(* CoDeSys 2.3 library: TcIoFunctions.lb6 *)
(* Libraries: STANDARD.LB6 5.6.98 12:03:02 *)

(* Data type *)
TYPE ST_KL1501InData :
STRUCT
	iState		: USINT;
	iDummy		: USINT;
	arrDataIn	: ARRAY[0..1] OF UINT;
END_STRUCT
END_TYPE

(* Data type *)
TYPE ST_KL1501OutData :
STRUCT
	iCtrl		: USINT;
	iDummy		: USINT;
	arrDataOut	: ARRAY[0..1] OF UINT;
END_STRUCT
END_TYPE

(* Data type *)
TYPE ST_KL27x1InData :
STRUCT
	iState		: USINT;
	iDummy		: USINT;
	iDataIn		: INT;
END_STRUCT
END_TYPE

(* Data type *)
TYPE ST_KL27x1OutData :
STRUCT
	iCtrl		: USINT;
	iDummy		: USINT;
	iDataOut	: INT;
END_STRUCT
END_TYPE

(* Data type *)
TYPE ST_KL3208InData :
STRUCT
	iState		: USINT;
	iDummy		: USINT;
	iDataIn		: INT;
END_STRUCT
END_TYPE

(* Data type *)
TYPE ST_KL3208OutData :
STRUCT
	iCtrl		: USINT;
	iDummy		: USINT;
	iDataOut	: INT;
END_STRUCT
END_TYPE

(* Data type *)
TYPE ST_KL320xInData :
STRUCT
	iState		: USINT;
	iDummy		: USINT;
	iDataIn		: INT;
END_STRUCT
END_TYPE

(* Data type *)
TYPE ST_KL320xOutData :
STRUCT
	iCtrl		: USINT;
	iDummy		: USINT;
	iDataOut	: INT;
END_STRUCT
END_TYPE

(* Data type *)
TYPE ST_KL3228InData :
STRUCT
	iState		: USINT;
	iDummy		: USINT;
	iDataIn		: INT;
END_STRUCT
END_TYPE

(* Data type *)
TYPE ST_KL3228OutData :
STRUCT
	iCtrl		: USINT;
	iDummy		: USINT;
	iDataOut	: INT;
END_STRUCT
END_TYPE

(* POU F_GetVersionTcIoFunctions, ST *)
FUNCTION F_GetVersionTcIoFunctions : UINT	(*Gets the library version info *)
VAR_INPUT
	nVersionElement		:	INT;
END_VAR
(*
	Possible nVersionElement parameter:
	1	:	major number
	2	:	minor number
	3	:	revision number
*)
VAR
END_VAR
(* Version history:
Date		|	Version	|	created with	|	Author		|	Remark
dd.mm.yyyy
-----------------------------------------------------------------------------------------------------------------------------------------------------------------------------------------------------------------
26.01.2016	|	1.0.0	|	TC 2.11 B2252	|	Peter S.  	|	first TC 2.11 release Folder K-Bus Terminals FB_KL1501Config, FB_KL27x1Config, FB_KL3208Config, FB_KL320xConfig, FB_KL3228Config;
*)	
CASE nVersionElement OF
1:	(* major number *)
	F_GetVersionTcIoFunctions := 1;
2:	(* minor number *)
	F_GetVersionTcIoFunctions := 0;
3:	(* revision number *)
	F_GetVersionTcIoFunctions := 0;
ELSE
	F_GetVersionTcIoFunctions := 16#FFFF;
END_CASE
END_FUNCTION

(* POU FB_KL1501Config, ST *)
FUNCTION_BLOCK FB_KL1501Config
VAR_INPUT
	bConfigurate			: BOOL; 		(*Rising edge starts configuration including read-configuration afterwards*)
	bReadConfig				: BOOL;			(*Rising edge reads the actual configuration*)
	iSetCounterType			: INT;			(*Counter-type to be set, see table*)
	bSetBackwardCounting	: BOOL;			(*Select backward-counting*)
	tTimeout				: TIME :=t#5s;	(*Time-out-time for Reading/Configuration - initially set to 5s*)
END_VAR
VAR_OUTPUT
	bBusy					: BOOL;			(*Reading or configuration is in progress*)
	bError					: BOOL;			(*Error while reading/configuration*)
	iErrorId				: UDINT;		(*Id of the last upcoming error*)
	iState					: USINT;		(*As long as the funcion-block is not busy, this variable shows the state of the terminal, otherwise it is 0*)
	iDataIn0				: UINT;			(*As long as the funcion-block is not busy, this variable shows the dataIn0 of the terminal, otherwise it keeps the value previous to reding/configuration*)
	iDataIn1				: UINT;			(*As long as the funcion-block is not busy, this variable shows the dataIn1 of the terminal, otherwise it keeps the value previous to reding/configuration*)
	iDataIn					: UDINT;		(*iDataIn1 and IDataIn0 put together as an UDINT, with iDataIn1 as High-Integer*)
	iTerminalType			: WORD;			(*Terminal-type-number, in this case 3228*)
	iSpecialType			: WORD;			(*Sub-type-number*)
	iFirmwareVersion		: WORD;			(*Firmware in ASCII-code*)
	sDescription			: STRING;		(*Terminal-type, special-type and firmware-version as readable text*)
	sCounterType			: STRING;		(*Text-description of entered counter-type*)
	bBackwardCounting		: BOOL;			(*TRUE: Backward-counting was selected*)
END_VAR
VAR
	rtRead					: R_TRIG;
	rtSet					: R_TRIG;
	bSetReq					: BOOL;
	tonTimeout				: TON;
	iStep					: INT;
	bSetConfigError			: BOOL;
	wReg32					: WORD;
	wSetReg32				: WORD;
	wFirmware				: WORD;
	pFirmware				: POINTER TO WORD;
	sFirmware				: STRING(2);
	iDataIn0Saved			: UINT;
	iDataIn1Saved			: UINT;
END_VAR
VAR_IN_OUT
	stInData   				: ST_KL1501InData;	(* Process image of the inputs. *)
	stOutData 				: ST_KL1501OutData;	(* Process image of the outputs. *)
END_VAR
tonTimeout	(PT:=tTimeout);
IF	tonTimeout.Q	THEN
	bError			:= TRUE;
	iErrorId		:= 16#8001;
	iStep			:= 0;
END_IF

rtSet	(CLK:=bConfigurate);
rtRead	(CLK:=bReadConfig);

IF	(rtSet.Q OR rtRead.Q)	AND NOT bBusy THEN
	bBusy			:= TRUE;
	bError			:= FALSE;
	iErrorId		:= 0;
	iDataIn0Saved	:= stInData.arrDataIn[0];
	iDataIn1Saved	:= stInData.arrDataIn[1];
	tonTimeout.IN	:= TRUE;
	iStep			:= 10;
	IF	rtSet.Q	THEN
		bSetReq	:= TRUE;
	END_IF
END_IF

IF bBusy THEN
	iDataIn0	:= iDataIn0Saved;
	iDataIn1	:= iDataIn1Saved;
	iState		:= 0;
ELSE
	iDataIn0	:= stInData.arrDataIn[0];
	iDataIn1	:= stInData.arrDataIn[1];
	iState		:= stInData.iState;
END_IF

iDataIn	:= UINT_TO_UDINT(iDataIn0)+(UINT_TO_UDINT(iDataIn1)*65536);

CASE iStep OF

0:	(*idle*)
	bBusy				:= FALSE;
	bSetReq				:= FALSE;
	tonTimeout.IN		:= FALSE;

10:	(*Klemmentyp (Kl32xx) auslesen: Register 8*)
	stOutData.iCtrl	:= 16#88;	(*Register 8 Lesen*)

	IF stInData.iState = 16#88 THEN
		iTerminalType	:= UINT_TO_WORD(stInData.arrDataIn[0]);
		iStep:=20;
	END_IF

20:	(*Spezialtyp (Kl1501-yyy) auslesen: Register 29*)
	stOutData.iCtrl	:= 16#9D;	(*Register 29 Lesen*)

	IF stInData.iState = 16#9D THEN
		iSpecialType	:= UINT_TO_WORD(stInData.arrDataIn[0]);
		iStep:=30;
	END_IF

30:	(*Firmware auslesen: Register 9*)
	stOutData.iCtrl	:= 16#89;	(*Register 9 Lesen*)

	IF stInData.iState = 16#89 THEN
		iFirmwareVersion:= UINT_TO_WORD(stInData.arrDataIn[0]);
		(*Umwandlung in STRING*)
		wFirmware		:= iFirmwareVersion;
		wFirmware		:= ROR(wFirmware,8);(*Reihenfolge der beiden Zeichen der Firmware tauschen*)
		pFirmware		:= ADR(sFirmware);	(*Einen Pointer auf den Info-String (Ausgang) legen*)
		pFirmware^		:= wFirmware;		(*Diesen Adressbereich mit dem richtig getauschen Wert beschreiben - damit ist auch der String beschrieben*)

		sDescription	:= CONCAT('Terminal ',WORD_TO_STRING(iTerminalType));

		CASE LEN(WORD_TO_STRING(iSpecialType)) OF
			1: sDescription	:= CONCAT(sDescription,'-000');
			2: sDescription	:= CONCAT(sDescription,'-00');
			3: sDescription	:= CONCAT(sDescription,'-0');
		ELSE
			sDescription	:= CONCAT(sDescription,'-');
		END_CASE

		sDescription	:= CONCAT(sDescription,WORD_TO_STRING(iSpecialType));
		sDescription	:= CONCAT(sDescription,' / Firmware ');
		sDescription	:= CONCAT(sDescription,sFirmware);

		IF bSetReq	THEN
			iStep:=100;
		ELSE
			iStep:=150;
		END_IF
	END_IF

	(*Falscher Klemmentyp angeschlossen, Konfiguration vorzeitig abbrechen*)
	IF (iTerminalType <> 1501)	THEN
		bError		:= TRUE;
		iErrorId	:= 16#8002;
		iStep		:= 160;
	END_IF
(*-----------------------------------------------------------------*)

100:(*jetzige Sensoreinstellung lesen: Register 32*)
	stOutData.iCtrl	:= 16#A0;	(*Register 32 Lesen*)

	IF stInData.iState = 16#A0 THEN
		wReg32			:= UINT_TO_WORD(stInData.arrDataIn[0]);
		A_SetConfigTable;			(*entsprechende Einstellungen vornehmen*)
		iStep:=110;
		IF	bSetConfigError	THEN
			iStep:=150;
		END_IF
	END_IF

110:(*Codewort Register 31 setzen: 16#1235 -> Schreibschutz aufheben*)
	stOutData.iCtrl	:= 16#DF;	(*Register 31 beschreiben*)
	stOutData.arrDataOut[0]	:= 16#1235;	(*Nutzdaten: Codewort*)

	IF stInData.iState = 16#9F THEN
		stOutData.iCtrl	:= 16#9F;	(*Register 31 Auslesen*)
		iStep:=120;
	END_IF

120:(*Bestätigung Codewort gesetzt erfragen*)
	IF	stInData.arrDataIn[0]	= 16#1235	THEN
		iStep:=130;
	END_IF

130:(*Nun Register 32 mit dem neuen Wert beschreiben*)
	stOutData.iCtrl	:= 16#E0;	(*Register 32 beschreiben*)
	stOutData.arrDataOut[0]	:= WORD_TO_UINT(wSetReg32);

	IF stInData.iState = 16#A0 THEN
		iStep:=140;
	END_IF

140:(*Codewort Register 31 löschen: 16#0000 -> Schreibschutz setzen*)
	stOutData.iCtrl	:= 16#DF;	(*Register 31 beschreiben*)
	stOutData.arrDataOut[0]	:= 16#0000;

	IF stInData.iState = 16#9F THEN
		iStep:=150;
	END_IF

150:(*nach erfolgter Parametrierung Sensoreinstellung lesen: Register 32*)
	stOutData.iCtrl	:= 16#A0;	(*Register 32 Lesen*)

	IF stInData.iState = 16#A0 THEN
		wReg32			:= UINT_TO_WORD(stInData.arrDataIn[0]);
		A_ReadConfigTable;
		iStep:=160;
	END_IF

160:(*Registerkommunikation beenden*)
	stOutData.iCtrl	:= 0; (*auch alle anderen Steuerbits mit ablöschen*)
	(*Rückmeldeabfrage Prozessdatenaustausch (Bit7) noch aktiv? *)
	(*alle anderen Bits könnten durch einen bestimmten Signalpegel gesetzt sein *)
	IF stInData.iState.7 = FALSE THEN
		iStep:=0;
	END_IF

END_CASE
END_FUNCTION_BLOCK
ACTION A_ReadConfigTable:
CASE (wReg32 AND 2#11100000000) OF	(*Check sensor-type via bits 8-10*)
	2#00100000000: sCounterType:='32-bit forward-backward-counter';
	2#01000000000: sCounterType:='Two 16-bit-forward-counter';
	2#10000000000: sCounterType:='32-bit gated forward-counter - Gate low inhibits';
	2#10100000000: sCounterType:='32-bit gated forward-counter - Gate high inhibits';
ELSE
	sCounterType:='Unknown';
	bError		:= TRUE;
	iErrorId	:= 16#8011;
END_CASE

bBackwardCounting:=wReg32.11;
END_ACTION
ACTION A_SetConfigTable:
bSetConfigError	:= FALSE;

wSetReg32:=wReg32 AND 2#1111000011111111;(*First clear the characteristical bits (8-11)*)

CASE iSetCounterType OF	(*Then set the counter-type via the bits 8-11*)

	0:	wSetReg32:=wSetReg32 OR 2#00100000000;(*32-bit forward-backward-counter*)
		wSetReg32.11:=bSetBackwardCounting;

	1:	wSetReg32:=wSetReg32 OR 2#01000000000;(*Two 16-bit-forward-counter*)
		wSetReg32.11:=bSetBackwardCounting;

	2:	wSetReg32:=wSetReg32 OR 2#10000000000;(*32-bit gated forward-counter - Gate low inhibits*)
		wSetReg32.11:=bSetBackwardCounting;

	3:	wSetReg32:=wSetReg32 OR 2#10100000000;(*32-bit gated forward-counter - Gate high inhibits*)
		wSetReg32.11:=bSetBackwardCounting;
ELSE
	bSetConfigError	:= TRUE;
	bError			:= TRUE;
	iErrorId		:= 16#8010;
END_CASE
END_ACTION

(* POU FB_KL27x1Config, ST *)
FUNCTION_BLOCK FB_KL27x1Config
VAR_INPUT
	bConfigurate			: BOOL; 		(*Rising edge starts configuration including read-configuration afterwards*)
	bReadConfig				: BOOL;			(*Rising edge reads the actual configuration*)
	bSetDimRampAbsolute		: BOOL;			(*FALSE: ramp-time refers to a step from 0..100%, TRUE: ramp-time refers to a step to the next value*)
	iSetRampTime			: INT;			(*Ramp-time to be set, see table*)
	bSetWatchdogDisable		: BOOL;			(*TRUE disables the watchdog for fieldbus-communication*)
	iSetWatchdogTimeout		: UINT;			(*Watchdog-time in 10ms-units*)
	iSetTimeoutOnValue		: UINT;			(*Value to be set, if timeout occurs and lamp was previously turned on*)
	iSetTimeoutOffValue		: UINT;			(*Value to be set, if timeout occurs and lamp was previously turned off*)
	iSetDimmerMode			: INT;			(*Dimmer-mode to be set, see table*)
	bSetOnAfterShortCircuit	: BOOL;			(*Selects, if the lamp has to be turned on after short-circuit*)
	bSetLineFrequency60Hz	: BOOL;			(*FALSE sets the line-frequency to 50Hz, TRUE to 60Hz*)
	tTimeout				: TIME :=t#5s;	(*Time-out-time for Reading/Configuration - initially set to 5s*)
END_VAR
VAR_OUTPUT
	bBusy					: BOOL;			(*Reading or configuration is in progress*)
	bError					: BOOL;			(*Error while reading/configuration*)
	iErrorId				: UDINT;		(*Id of the last upcoming error*)
	iState					: USINT;		(*As long as the funcion-block is not busy, this variable shows the state of the terminal, otherwise it is 0*)
	iTerminalType			: WORD;			(*Terminal-type-number, e.g. 2751*)
	iSpecialType			: WORD;			(*Sub-type-number*)
	iFirmwareVersion		: WORD;			(*Firmware in ASCII-code*)
	sDescription			: STRING;		(*Terminal-type, special-type and firmware-version as readable text*)

	bDimRampAbsolute		: BOOL;			(*TRUE: Dimramp was set to absolute - FALSE Dimramp was set to relative*)
	sRampTime				: STRING;		(*Ramp-time, which was set, according to the table*)
	bWatchdogDisable		: BOOL;			(*TRUE: Watchdog was disabled*)
	tWatchdogTimeout		: TIME;			(*Entered Watchdog-time*)
	iTimeoutOnValue			: UINT;			(*Timeout on-value, which was set*)
	iTimeoutOffValue		: UINT;			(*Timeout off-value, which was set*)
	sDimmerMode				: STRING;		(*Dimmer-mode, which was selected*)
	sAfterShortCircuit		: STRING;		(*Selected behaviour after short-circuit - on or off*)
	sLineFrequency			: STRING;		(*Selected line-frequency - 50 or 60 Hz*)
END_VAR
VAR
	rtRead					: R_TRIG;
	rtSet					: R_TRIG;
	bSetReq					: BOOL;
	tonTimeout				: TON;
	iStep					: INT;
	bSetConfigError			: BOOL;
	wReg32					: WORD;
	wSetReg32				: WORD;
	wReg35					: WORD;
	wSetReg35				: WORD;
	wReg36					: WORD;
	wSetReg36				: WORD;
	wReg37					: WORD;
	wSetReg37				: WORD;
	wReg38					: WORD;
	wSetReg38				: WORD;
	wReg39					: WORD;
	wSetReg39				: WORD;
	wReg40					: WORD;
	wSetReg40				: WORD;
	wReg41					: WORD;
	wSetReg41				: WORD;
	wFirmware				: WORD;
	pFirmware				: POINTER TO WORD;
	sFirmware				: STRING(2);
END_VAR
VAR_IN_OUT
	stInData   				: ST_KL27x1InData;	(* Process image of the inputs. *)
	stOutData 				: ST_KL27x1OutData;	(* Process image of the outputs. *)
END_VAR
tonTimeout	(PT:=tTimeout);
IF	tonTimeout.Q	THEN
	bError			:= TRUE;
	iErrorId		:= 16#8001;
	iStep			:= 0;
END_IF

rtSet	(CLK:=bConfigurate);
rtRead	(CLK:=bReadConfig);

IF	(rtSet.Q OR rtRead.Q)	AND NOT bBusy THEN
	bBusy			:= TRUE;
	bError			:= FALSE;
	iErrorId		:= 0;
	tonTimeout.IN	:= TRUE;
	iStep			:= 10;
	IF	rtSet.Q	THEN
		bSetReq	:= TRUE;
	END_IF
END_IF

IF bBusy THEN
	iState		:= 0;
ELSE
	iState		:= stInData.iState;
END_IF


CASE iStep OF

0:	(*idlde*)
	bBusy				:= FALSE;
	bSetReq				:= FALSE;
	tonTimeout.IN		:= FALSE;

10:	(*Klemmentyp (Kl27xx) auslesen: Register 8*)
	stOutData.iCtrl	:= 16#88;	(*Register 8 Lesen*)

	IF stInData.iState = 16#88 THEN
		iTerminalType	:= INT_TO_WORD(stInData.iDataIn);
		iStep:=20;
	END_IF

20:	(*Spezialtyp (Kl27xx-yyy) auslesen: Register 29*)
	stOutData.iCtrl	:= 16#9D;	(*Register 29 Lesen*)

	IF stInData.iState = 16#9D THEN
		iSpecialType	:= INT_TO_WORD(stInData.iDataIn);
		iStep:=30;
	END_IF

30:	(*Firmware auslesen: Register 9*)
	stOutData.iCtrl	:= 16#89;	(*Register 9 Lesen*)

	IF stInData.iState = 16#89 THEN
		iFirmwareVersion:= INT_TO_WORD(stInData.iDataIn);
		(*Umwandlung in STRING*)
		wFirmware		:= iFirmwareVersion;
		wFirmware		:= ROR(wFirmware,8);(*Reihenfolge der beiden Zeichen der Firmware tauschen*)
		pFirmware		:= ADR(sFirmware);	(*Einen Pointer auf den Info-String (Ausgang) legen*)
		pFirmware^		:= wFirmware;		(*Diesen Adressbereich mit dem richtig getauschen Wert beschreiben - damit ist auch der String beschrieben*)

		sDescription	:= CONCAT('Terminal ',WORD_TO_STRING(iTerminalType));

		CASE LEN(WORD_TO_STRING(iSpecialType)) OF
			1: sDescription	:= CONCAT(sDescription,'-000');
			2: sDescription	:= CONCAT(sDescription,'-00');
			3: sDescription	:= CONCAT(sDescription,'-0');
		ELSE
			sDescription	:= CONCAT(sDescription,'-');
		END_CASE

		sDescription	:= CONCAT(sDescription,WORD_TO_STRING(iSpecialType));
		sDescription	:= CONCAT(sDescription,' / Firmware ');
		sDescription	:= CONCAT(sDescription,sFirmware);

		IF bSetReq	THEN
			iStep:=100;
		ELSE
			iStep:=150;
		END_IF
	END_IF

	(*Falscher Klemmentyp angeschlossen, Konfiguration vorzeitig abbrechen*)
	IF ((iTerminalType <> 2751)	AND (iTerminalType <> 2761))	THEN
		bError		:= TRUE;
		iErrorId	:= 16#8002;
		iStep		:= 160;
	END_IF

(*-----------------------------------------------------------------*)

100:(*jetzige Sensoreinstellung lesen: Register 32*)
	stOutData.iCtrl	:= 16#A0;	(*Register 32 Lesen*)

	IF stInData.iState = 16#A0 THEN
		wReg32			:= INT_TO_WORD(stInData.iDataIn);
		A_SetConfigTable;			(*entsprechende Einstellungen vornehmen*)
		iStep:=110;
		IF	bSetConfigError	THEN
			iStep:=150;
		END_IF
	END_IF

110:(*Codewort Register 31 setzen: 16#1235 -> Schreibschutz aufheben*)
	stOutData.iCtrl	:= 16#DF;	(*Register 31 beschreiben*)
	stOutData.iDataOut	:= 16#1235;	(*Nutzdaten: Codewort*)

	IF stInData.iState = 16#9F THEN
		stOutData.iCtrl	:= 16#9F;	(*Register 31 Auslesen*)
		iStep:=120;
	END_IF

120:(*Bestätigung Codewort gesetzt erfragen*)
	IF	stInData.iDataIn	= 16#1235	THEN
		iStep:=130;
	END_IF

130:(*Register 32 mit dem neuen Wert beschreiben*)
	stOutData.iCtrl	:= 16#E0;	(*Register 32 beschreiben*)
	stOutData.iDataOut	:= WORD_TO_INT(wSetReg32);

	IF stInData.iState = 16#A0 THEN
		iStep:=131;
	END_IF

131:(*Register 35 mit dem neuen Wert beschreiben*)
	stOutData.iCtrl	:= 16#E3;	(*Register 35 beschreiben*)
	stOutData.iDataOut	:= WORD_TO_INT(wSetReg35);

	IF stInData.iState = 16#A3 THEN
		iStep:=132;
	END_IF

132:(*Register 36 mit dem neuen Wert beschreiben*)
	stOutData.iCtrl	:= 16#E4;	(*Register 36 beschreiben*)
	stOutData.iDataOut	:= WORD_TO_INT(wSetReg36);

	IF stInData.iState = 16#A4 THEN
		iStep:=133;
	END_IF

133:(*Register 37 mit dem neuen Wert beschreiben*)
	stOutData.iCtrl	:= 16#E5;	(*Register 37 beschreiben*)
	stOutData.iDataOut	:= WORD_TO_INT(wSetReg37);

	IF stInData.iState = 16#A5 THEN
		iStep:=134;
	END_IF

134:(*Register 38 mit dem neuen Wert beschreiben*)
	stOutData.iCtrl	:= 16#E6;	(*Register 38 beschreiben*)
	stOutData.iDataOut	:= WORD_TO_INT(wSetReg38);

	IF stInData.iState = 16#A6 THEN
		iStep:=135;
	END_IF

135:(*Register 39 mit dem neuen Wert beschreiben*)
	stOutData.iCtrl	:= 16#E7;	(*Register 39 beschreiben*)
	stOutData.iDataOut	:= WORD_TO_INT(wSetReg39);

	IF stInData.iState = 16#A7 THEN
		iStep:=136;
	END_IF

136:(*Register 40 mit dem neuen Wert beschreiben*)
	stOutData.iCtrl	:= 16#E8;	(*Register 40 beschreiben*)
	stOutData.iDataOut	:= WORD_TO_INT(wSetReg40);

	IF stInData.iState = 16#A8 THEN
		iStep:=137;
	END_IF

137:(*Register 41 mit dem neuen Wert beschreiben*)
	stOutData.iCtrl	:= 16#E9;	(*Register 41 beschreiben*)
	stOutData.iDataOut	:= WORD_TO_INT(wSetReg41);

	IF stInData.iState = 16#A9 THEN
		iStep:=140;
	END_IF

140:(*Codewort Register 31 löschen: 16#0000 -> Schreibschutz setzen*)
	stOutData.iCtrl	:= 16#DF;	(*Register 31 beschreiben*)
	stOutData.iDataOut	:= 16#0000;

	IF stInData.iState = 16#9F THEN
		iStep:=150;
	END_IF

150:(*nach erfolgter Parametrierung Konfiguration lesen: Register 32*)
	stOutData.iCtrl	:= 16#A0;	(*Register 32 Lesen*)

	IF stInData.iState = 16#A0 THEN
		wReg32			:= INT_TO_WORD(stInData.iDataIn);
		iStep:=151;
	END_IF

151:(*nach erfolgter Parametrierung Konfiguration lesen: Register 35*)
	stOutData.iCtrl	:= 16#A3;	(*Register 35 Lesen*)

	IF stInData.iState = 16#A3 THEN
		wReg35			:= INT_TO_WORD(stInData.iDataIn);
		iStep:=152;
	END_IF

152:(*nach erfolgter Parametrierung Konfiguration lesen: Register 36*)
	stOutData.iCtrl	:= 16#A4;	(*Register 36 Lesen*)

	IF stInData.iState = 16#A4 THEN
		wReg36			:= INT_TO_WORD(stInData.iDataIn);
		iStep:=153;
	END_IF

153:(*nach erfolgter Parametrierung Konfiguration lesen: Register 37*)
	stOutData.iCtrl	:= 16#A5;	(*Register 37 Lesen*)

	IF stInData.iState = 16#A5 THEN
		wReg37			:= INT_TO_WORD(stInData.iDataIn);
		iStep:=154;
	END_IF

154:(*nach erfolgter Parametrierung Konfiguration lesen: Register 38*)
	stOutData.iCtrl	:= 16#A6;	(*Register 38 Lesen*)

	IF stInData.iState = 16#A6 THEN
		wReg38			:= INT_TO_WORD(stInData.iDataIn);
		iStep:=155;
	END_IF

155:(*nach erfolgter Parametrierung Konfiguration lesen: Register 39*)
	stOutData.iCtrl	:= 16#A7;	(*Register 39 Lesen*)

	IF stInData.iState = 16#A7 THEN
		wReg39			:= INT_TO_WORD(stInData.iDataIn);
		iStep:=156;
	END_IF

156:(*nach erfolgter Parametrierung Konfiguration lesen: Register 40*)
	stOutData.iCtrl	:= 16#A8;	(*Register 40 Lesen*)

	IF stInData.iState = 16#A8 THEN
		wReg40			:= INT_TO_WORD(stInData.iDataIn);
		iStep:=157;
	END_IF


157:(*nach erfolgter Parametrierung Konfiguration lesen: Register 41*)
	stOutData.iCtrl	:= 16#A9;	(*Register 41 Lesen*)

	IF stInData.iState = 16#A9 THEN
		wReg41			:= INT_TO_WORD(stInData.iDataIn);
		A_ReadConfigTable;
		iStep:=160;
	END_IF


160:(*Registerkommunikation beenden*)
	stOutData.iCtrl	:= 0; (*auch alle anderen Steuerbits mit ablöschen*)
	(*Rückmeldeabfrage Prozessdatenaustausch (Bit7) noch aktiv? *)
	(*alle anderen Bits könnten durch einen bestimmten Signalpegel gesetzt sein *)
	IF stInData.iState.7 = FALSE THEN
		iStep:=0;
	END_IF

END_CASE
END_FUNCTION_BLOCK
ACTION A_ReadConfigTable:
bWatchdogDisable	:= wReg32.2;
bDimRampAbsolute	:= wReg32.3;


CASE wReg35 OF
	0:	sRampTime	:= '50 ms';
	1:	sRampTime	:= '100 ms';
	2:	sRampTime	:= '200 ms';
	3:	sRampTime	:= '500 ms';
	4:	sRampTime	:= '1 s';
	5:	sRampTime	:= '2 s';
	6:	sRampTime	:= '5 s';
	7:	sRampTime	:= '10 s';
ELSE
	sRampTime	:= 'unknown register-entry';
	bError		:= TRUE;
	iErrorId	:= 16#801A;
END_CASE


tWatchdogTimeout	:= WORD_TO_TIME(wReg36)*10;
iTimeoutOnValue		:= wReg37;
iTimeoutOffValue	:= wReg38;


CASE wReg39 OF
	0:	sDimmerMode	:= '0 - Automatic recognition';
	1:	sDimmerMode	:= '1 - Trailing phase angle';
	2:	sDimmerMode	:= '2 - Leading phase angle';
	3:	sDimmerMode	:= '3 - Rectifier mode, positive';
	4:	sDimmerMode	:= '4 - Rectifier mode, negative';
ELSE
	sDimmerMode	:= 'unknown register-entry';
	bError		:= TRUE;
	iErrorId	:= 16#801B;
END_CASE


CASE wReg40 OF
	0:	sAfterShortCircuit := 'Off';
	1:	sAfterShortCircuit := 'On';
ELSE
	sAfterShortCircuit	:= 'unknown register-entry';
	bError				:= TRUE;
	iErrorId			:= 16#801C;
END_CASE


CASE wReg41 OF
	0:	sLineFrequency := '50 Hz';
	1:	sLineFrequency := '60 Hz';
ELSE
	sLineFrequency	:= 'unknown register-entry';
	bError			:= TRUE;
	iErrorId		:= 16#801D;
END_CASE
END_ACTION
ACTION A_SetConfigTable:
bSetConfigError	:= FALSE;

wSetReg32	:= wReg32	AND 2#1111111111110011;(*Clear bits 2 and 3 of Reg32*)
wSetReg32.2	:= bSetWatchdogDisable;
wSetReg32.3	:= bSetDimRampAbsolute;

CASE iSetRampTime OF
	0:	wSetReg35	:= 0;		(*50 ms*)
	1:	wSetReg35	:= 1;		(*100 ms*)
	2:	wSetReg35	:= 2;		(*200 ms*)
	3:	wSetReg35	:= 3;		(*500 ms*)
	4:	wSetReg35	:= 4;		(*1 s*)
	5:	wSetReg35	:= 5;		(*2 s*)
	6:	wSetReg35	:= 6;		(*5 s*)
	7:	wSetReg35	:= 7;		(*10 s*)
ELSE
	bSetConfigError	:= TRUE;
	bError			:= TRUE;
	iErrorId		:= 16#8018;
END_CASE


wSetReg36	:=	UINT_TO_WORD(iSetWatchdogTimeout);
wSetReg37	:=	UINT_TO_WORD(iSetTimeoutOnValue);
wSetReg38	:=	UINT_TO_WORD(iSetTimeoutOffValue);


CASE iSetDimmerMode OF
	0:	wSetReg39	:= 0;		(*automatic recognition*)
	1:	wSetReg39	:= 1;		(*trailing phase angle*)
	2:	wSetReg39	:= 2;		(*leading phase angle*)
	3:	wSetReg39	:= 3;		(*Rectifier mode, positive*)
	4:	wSetReg39	:= 4;		(*Rectifier mode, negative*)
ELSE
	bSetConfigError	:= TRUE;
	bError			:= TRUE;
	iErrorId		:= 16#8019;
END_CASE

IF	bSetOnAfterShortCircuit	THEN
		wSetReg40	:= 1;
ELSE	wSetReg40	:= 0;
END_IF

IF	bSetLineFrequency60Hz	THEN
		wSetReg41	:= 1;
ELSE	wSetReg41	:= 0;
END_IF
END_ACTION

(* POU FB_KL3208Config, ST *)
FUNCTION_BLOCK FB_KL3208Config
VAR_INPUT
	bConfigurate		: BOOL; 		(*Rising edge starts configuration including read-configuration afterwards*)
	bReadConfig			: BOOL;			(*Rising edge reads the actual configuration*)
	iSetSensorType		: INT;			(*Sensor-type to be set, see table*)
	tTimeout			: TIME :=t#5s;	(*Time-out-time for Reading/Configuration - initially set to 5s*)
END_VAR
VAR_OUTPUT
	bBusy				: BOOL;			(*Reading or configuration is in progress*)
	bError				: BOOL;			(*Error while reading/configuration*)
	iErrorId			: UDINT;		(*Id of the last upcoming error*)
	iState				: USINT;		(*As long as the funcion-block is not busy, this variable shows the state of the terminal, otherwise it is 0*)
	iDataIn				: INT;			(*As long as the funcion-block is not busy, this variable shows the dataIn of the terminal, otherwise it keeps the value previous to reding/configuration*)
	iTerminalType		: WORD;			(*Terminal-type-number, in this case 3208*)
	iSpecialType		: WORD;			(*Sub-type-number*)
	iFirmwareVersion	: WORD;			(*Firmware in ASCII-code*)
	sDescription		: STRING;		(*Terminal-type, special-type and firmware-version as readable text*)
	sSensorType			: STRING;		(*Text-description of entered sensor-type*)
END_VAR
VAR
	rtRead				: R_TRIG;
	rtSet				: R_TRIG;
	bSetReq				: BOOL;
	tonTimeout			: TON;
	iStep				: INT;
	bSetConfigError		: BOOL;
	wReg32				: WORD;
	wSetReg32			: WORD;
	wReg39				: WORD;
	wSetReg39			: WORD;
	wFirmware			: WORD;
	pFirmware			: POINTER TO WORD;
	sFirmware			: STRING(2);
	iDataInSaved		: INT;
END_VAR
VAR_IN_OUT
	stInData   			: ST_KL3208InData;	(* Process image of the inputs. *)
	stOutData 			: ST_KL3208OutData;	(* Process image of the outputs. *)
END_VAR
tonTimeout	(PT:=tTimeout);
IF	tonTimeout.Q	THEN
	bError			:= TRUE;
	iErrorId		:= 16#8001;
	iStep			:= 0;
END_IF

rtSet	(CLK:=bConfigurate);
rtRead	(CLK:=bReadConfig);

IF	(rtSet.Q OR rtRead.Q)	AND NOT bBusy THEN
	bBusy			:= TRUE;
	bError			:= FALSE;
	iErrorId		:= 0;
	iDataInSaved	:= stInData.iDataIn;
	tonTimeout.IN	:= TRUE;
	iStep			:= 10;
	IF	rtSet.Q	THEN
		bSetReq	:= TRUE;
	END_IF
END_IF

IF bBusy THEN
	iDataIn		:= iDataInSaved;
	iState		:= 0;
ELSE
	iDataIn		:= stInData.iDataIn;
	iState		:= stInData.iState;
END_IF


CASE iStep OF

0:	(*idle*)
	bBusy				:= FALSE;
	bSetReq				:= FALSE;
	tonTimeout.IN		:= FALSE;

10:	(*Klemmentyp (Kl32xx) auslesen: Register 8*)
	stOutData.iCtrl	:= 16#88;	(*Register 8 Lesen*)

	IF stInData.iState = 16#88 THEN
		iTerminalType	:= INT_TO_WORD(stInData.iDataIn);
		iStep:=20;
	END_IF

20:	(*Spezialtyp (Kl32xx-yyy) auslesen: Register 29*)
	stOutData.iCtrl	:= 16#9D;	(*Register 29 Lesen*)

	IF stInData.iState = 16#9D THEN
		iSpecialType	:= INT_TO_WORD(stInData.iDataIn);
		iStep:=30;
	END_IF

30:	(*Firmware auslesen: Register 9*)
	stOutData.iCtrl	:= 16#89;	(*Register 9 Lesen*)

	IF stInData.iState = 16#89 THEN
		iFirmwareVersion:= INT_TO_WORD(stInData.iDataIn);
		(*Umwandlung in STRING*)
		wFirmware		:= iFirmwareVersion;
		wFirmware		:= ROR(wFirmware,8);(*Reihenfolge der beiden Zeichen der Firmware tauschen*)
		pFirmware		:= ADR(sFirmware);	(*Einen Pointer auf den Info-String (Ausgang) legen*)
		pFirmware^		:= wFirmware;		(*Diesen Adressbereich mit dem richtig getauschen Wert beschreiben - damit ist auch der String beschrieben*)

		sDescription	:= CONCAT('Terminal ',WORD_TO_STRING(iTerminalType));

		CASE LEN(WORD_TO_STRING(iSpecialType)) OF
			1: sDescription	:= CONCAT(sDescription,'-000');
			2: sDescription	:= CONCAT(sDescription,'-00');
			3: sDescription	:= CONCAT(sDescription,'-0');
		ELSE
			sDescription	:= CONCAT(sDescription,'-');
		END_CASE

		sDescription	:= CONCAT(sDescription,WORD_TO_STRING(iSpecialType));
		sDescription	:= CONCAT(sDescription,' / Firmware ');
		sDescription	:= CONCAT(sDescription,sFirmware);

		IF bSetReq	THEN
			iStep:=100;
		ELSE
			iStep:=150;
		END_IF
	END_IF

	(*Falscher Klemmentyp angeschlossen, Konfiguration vorzeitig abbrechen*)
	IF (iTerminalType <> 3208)	THEN
		bError		:= TRUE;
		iErrorId	:= 16#8002;
		iStep		:= 160;
	END_IF

(*-----------------------------------------------------------------*)

100:(*jetzige Sensoreinstellung lesen: Register 32*)
	stOutData.iCtrl	:= 16#A0;	(*Register 32 Lesen*)

	IF stInData.iState = 16#A0 THEN
		wReg32			:= INT_TO_WORD(stInData.iDataIn);
		iStep:=105;
	END_IF

105:(*jetzige Sensoreinstellung lesen: Register 39*)
	stOutData.iCtrl	:= 16#A7;	(*Register 39 Lesen*)

	IF stInData.iState = 16#A7 THEN
		wReg39			:= INT_TO_WORD(stInData.iDataIn);
		A_SetConfigTable;			(*entsprechende Einstellungen vornehmen*)
		iStep:=110;
		IF	bSetConfigError	THEN
			iStep:=150;
		END_IF
	END_IF

110:(*Codewort Register 31 setzen: 16#1235 -> Schreibschutz aufheben*)
	stOutData.iCtrl	:= 16#DF;	(*Register 31 beschreiben*)
	stOutData.iDataOut	:= 16#1235;	(*Nutzdaten: Codewort*)

	IF stInData.iState = 16#9F THEN
		stOutData.iCtrl	:= 16#9F;	(*Register 31 Auslesen*)
		iStep:=120;
	END_IF

120:(*Bestätigung Codewort gesetzt erfragen*)
	IF	stInData.iDataIn	= 16#1235	THEN
		iStep:=130;
	END_IF

130:(*Nun Register 32 mit dem neuen Wert beschreiben*)
	stOutData.iCtrl	:= 16#E0;	(*Register 32 beschreiben*)
	stOutData.iDataOut	:= WORD_TO_INT(wSetReg32);

	IF stInData.iState = 16#A0 THEN
		iStep:=135;
	END_IF

135:(*Und Register 39 mit dem neuen Wert beschreiben*)
	stOutData.iCtrl	:= 16#E7;	(*Register 39 beschreiben*)
	stOutData.iDataOut	:= WORD_TO_INT(wSetReg39);

	IF stInData.iState = 16#A7 THEN
		iStep:=140;
	END_IF

140:(*Codewort Register 31 löschen: 16#0000 -> Schreibschutz setzen*)
	stOutData.iCtrl	:= 16#DF;	(*Register 31 beschreiben*)
	stOutData.iDataOut	:= 16#0000;

	IF stInData.iState = 16#9F THEN
		iStep:=150;
	END_IF

150:(*nach erfolgter Parametrierung Sensoreinstellung lesen: Register 32*)
	stOutData.iCtrl	:= 16#A0;	(*Register 32 Lesen*)

	IF stInData.iState = 16#A0 THEN
		wReg32			:= INT_TO_WORD(stInData.iDataIn);
		iStep:=155;
	END_IF

155:(*nach erfolgter Parametrierung Sensoreinstellung lesen: Register 39*)
	stOutData.iCtrl	:= 16#A7;	(*Register 39 Lesen*)

	IF stInData.iState = 16#A7 THEN
		wReg39			:= INT_TO_WORD(stInData.iDataIn);
		A_ReadConfigTable;
		iStep:=160;
	END_IF

160:(*Registerkommunikation beenden*)
	stOutData.iCtrl	:= 0; (*auch alle anderen Steuerbits mit ablöschen*)
	(*Rückmeldeabfrage Prozessdatenaustausch (Bit7) noch aktiv? *)
	(*alle anderen Bits könnten durch einen bestimmten Signalpegel gesetzt sein *)
	IF stInData.iState.7 = FALSE THEN
		iStep:=0;
	END_IF

END_CASE
END_FUNCTION_BLOCK
ACTION A_ReadConfigTable:
(*IF Reg39 is set to 0, Reg32 is responsible for the sensor-type, otherwise Reg39 sets the sensor*)

IF	wReg39=0	THEN
	CASE (SHR(wReg32,12)) OF	(*Check sensor-type via the 4 most significant bits*)
		2#0000: sSensorType	:= 'PT1000';
		2#0001: sSensorType	:= 'NI1000';
		2#0010: sSensorType	:= 'RSNI1000';
	ELSE
		sSensorType	:='Unknown';
		bError		:= TRUE;
		iErrorId	:= 16#8021;
	END_CASE
ELSE
	CASE wReg39 OF
		16#32: sSensorType	:= 'NCT1K8';
		16#33: sSensorType	:= 'NCT1K8_TK';
		16#34: sSensorType	:= 'NCT2K2';
		16#35: sSensorType	:= 'NCT3K';
		16#36: sSensorType	:= 'NCT5K';
		16#37: sSensorType	:= 'NTC10K';
		16#38: sSensorType	:= 'NTC10KPRE';
		16#39: sSensorType	:= 'NTC10K_3204';
		16#3A: sSensorType	:= 'NTC10KTYP2';
		16#3B: sSensorType	:= 'NTC10KTYP3';
		16#3C: sSensorType	:= 'NTC10KDALE';
		16#3D: sSensorType	:= 'NTC10K3A221';
		16#3E: sSensorType	:= 'NTC20K';
		16#64: sSensorType	:= 'Poti, Resolution 0,1 Ohm';
		16#65: sSensorType	:= 'Poti, Resolution 1 Ohm';
		16#C8: sSensorType	:= 'NTC100K';
		16#FF: sSensorType	:= 'User defined';
	ELSE
		sSensorType	:='Unknown';
		bError		:= TRUE;
		iErrorId	:= 16#8021;
	END_CASE
END_IF
END_ACTION
ACTION A_SetConfigTable:
bSetConfigError	:= FALSE;

CASE iSetSensorType OF	(*Then set the sensor-type via the 4 most significant bits*)

	0:	wSetReg32	:= wReg32		AND 2#0000111111111111;(*First clear the first 4 bits*)
		wSetReg32	:= wSetReg32	OR 2#0000000000000000;(*PT1000*)	(*Then set the sensor-type via the 4 most significant bits*)
		wSetReg39	:= 0;

	1:	wSetReg32	:= wReg32		AND 2#0000111111111111;(*First clear the first 4 bits*)
		wSetReg32	:= wSetReg32	OR 2#0001000000000000;(*NI1000*)	(*Then set the sensor-type via the 4 most significant bits*)
		wSetReg39	:= 0;

	2:	wSetReg32	:= wReg32		AND 2#0000111111111111;(*First clear the first 4 bits*)
		wSetReg32	:= wSetReg32	OR 2#0010000000000000;(*RSNI1000*)	(*Then set the sensor-type via the 4 most significant bits*)
		wSetReg39	:= 0;


	3:	wSetReg39	:= 16#32;		(*NCT1K8*)
	4:	wSetReg39	:= 16#33;		(*NCT1K8_TK*)
	5:	wSetReg39	:= 16#34;		(*NCT2K2*)
	6:	wSetReg39	:= 16#35;		(*NCT3K*)
	7:	wSetReg39	:= 16#36;		(*NCT5K*)
	8:	wSetReg39	:= 16#37;		(*NTC10K*)
	9:	wSetReg39	:= 16#38;		(*NTC10KPRE*)
	10:	wSetReg39	:= 16#39;		(*NTC10K_3204*)
	11:	wSetReg39	:= 16#3A;		(*NTC10KTYP2*)
	12:	wSetReg39	:= 16#3B;		(*NTC10KTYP3*)
	13:	wSetReg39	:= 16#3C;		(*NTC10KDALE*)
	14:	wSetReg39	:= 16#3D;		(*NTC10K3A221*)
	15:	wSetReg39	:= 16#3E;		(*NTC20K*)
	16:	wSetReg39	:= 16#64;		(*Poti, Resolution 0,1 Ohm*)
	17:	wSetReg39	:= 16#65;		(*Poti, Resolution 1 Ohm*)
	18:	wSetReg39	:= 16#C8;		(*NTC100K*)
ELSE
	bSetConfigError	:= TRUE;
	bError			:= TRUE;
	iErrorId		:= 16#8020;
END_CASE
END_ACTION

(* POU FB_KL320xConfig, ST *)
FUNCTION_BLOCK FB_KL320xConfig
VAR_INPUT
	bConfigurate		: BOOL; 		(*Rising edge starts configuration including read-configuration afterwards*)
	bReadConfig			: BOOL;			(*Rising edge reads the actual configuration*)
	iSetSensorType		: INT;			(*Sensor-type to be set, see table*)
	tTimeout			: TIME :=t#5s;	(*Time-out-time for Reading/Configuration - initially set to 5s*)
END_VAR
VAR_OUTPUT
	bBusy				: BOOL;			(*Reading or configuration is in progress*)
	bError				: BOOL;			(*Error while reading/configuration*)
	iErrorId			: UDINT;		(*Id of the last upcoming error*)
	iState				: USINT;		(*As long as the funcion-block is not busy, this variable shows the state of the terminal, otherwise it is 0*)
	iDataIn				: INT;			(*As long as the funcion-block is not busy, this variable shows the dataIn of the terminal, otherwise it keeps the value previous to reding/configuration*)
	iTerminalType		: WORD;			(*Terminal-type-number, e.g. 3204*)
	iSpecialType		: WORD;			(*Sub-type-number*)
	iFirmwareVersion	: WORD;			(*Firmware in ASCII-code*)
	sDescription		: STRING;		(*Terminal-type, special-type and firmware-version as readable text*)
	sSensorType			: STRING;		(*Text-description of entered sensor-type*)
	bTwoWiredConnection	: BOOL;			(*Shows, if two-wired connection is selected*)
END_VAR
VAR
	rtRead				: R_TRIG;
	rtSet				: R_TRIG;
	bSetReq				: BOOL;
	tonTimeout			: TON;
	iStep				: INT;
	bSetConfigError		: BOOL;
	wReg32				: WORD;
	wSetReg32			: WORD;
	wFirmware			: WORD;
	pFirmware			: POINTER TO WORD;
	sFirmware			: STRING(2);
	iDataInSaved		: INT;
END_VAR
VAR_IN_OUT
	stInData   			: ST_KL320xInData;	(* Process image of the inputs. *)
	stOutData 			: ST_KL320xOutData;	(* Process image of the outputs. *)
END_VAR
tonTimeout	(PT:=tTimeout);
IF	tonTimeout.Q	THEN
	bError			:= TRUE;
	iErrorId		:= 16#8001;
	iStep			:= 0;
END_IF

rtSet	(CLK:=bConfigurate);
rtRead	(CLK:=bReadConfig);

IF	(rtSet.Q OR rtRead.Q)	AND NOT bBusy THEN
	bBusy			:= TRUE;
	bError			:= FALSE;
	iErrorId		:= 0;
	iDataInSaved	:= stInData.iDataIn;
	tonTimeout.IN	:= TRUE;
	iStep			:= 10;
	IF	rtSet.Q	THEN
		bSetReq	:= TRUE;
	END_IF
END_IF

IF bBusy THEN
	iDataIn		:= iDataInSaved;
	iState		:= 0;
ELSE
	iDataIn		:= stInData.iDataIn;
	iState		:= stInData.iState;
END_IF


CASE iStep OF

0:	(*idle*)
	bBusy				:= FALSE;
	bSetReq				:= FALSE;
	tonTimeout.IN		:= FALSE;

10:	(*Klemmentyp (Kl32xx) auslesen: Register 8*)
	stOutData.iCtrl	:= 16#88;	(*Register 8 Lesen*)

	IF stInData.iState = 16#88 THEN
		iTerminalType	:= INT_TO_WORD(stInData.iDataIn);
		iStep:=20;
	END_IF

20:	(*Spezialtyp (Kl32xx-yyy) auslesen: Register 29*)
	stOutData.iCtrl	:= 16#9D;	(*Register 29 Lesen*)

	IF stInData.iState = 16#9D THEN
		iSpecialType	:= INT_TO_WORD(stInData.iDataIn);
		iStep:=30;
	END_IF

30:	(*Firmware auslesen: Register 9*)
	stOutData.iCtrl	:= 16#89;	(*Register 9 Lesen*)

	IF stInData.iState = 16#89 THEN
		iFirmwareVersion:= INT_TO_WORD(stInData.iDataIn);
		(*Umwandlung in STRING*)
		wFirmware		:= iFirmwareVersion;
		wFirmware		:= ROR(wFirmware,8);(*Reihenfolge der beiden Zeichen der Firmware tauschen*)
		pFirmware		:= ADR(sFirmware);	(*Einen Pointer auf den Info-String (Ausgang) legen*)
		pFirmware^		:= wFirmware;		(*Diesen Adressbereich mit dem richtig getauschen Wert beschreiben - damit ist auch der String beschrieben*)

		sDescription	:= CONCAT('Terminal ',WORD_TO_STRING(iTerminalType));

		CASE LEN(WORD_TO_STRING(iSpecialType)) OF
			1: sDescription	:= CONCAT(sDescription,'-000');
			2: sDescription	:= CONCAT(sDescription,'-00');
			3: sDescription	:= CONCAT(sDescription,'-0');
		ELSE
			sDescription	:= CONCAT(sDescription,'-');
		END_CASE

		sDescription	:= CONCAT(sDescription,WORD_TO_STRING(iSpecialType));
		sDescription	:= CONCAT(sDescription,' / Firmware ');
		sDescription	:= CONCAT(sDescription,sFirmware);

		IF bSetReq	THEN
			iStep:=100;
		ELSE
			iStep:=150;
		END_IF
	END_IF

	(*Falscher Klemmentyp angeschlossen, Konfiguration vorzeitig abbrechen*)
	IF ((iTerminalType <> 3201)	AND (iTerminalType <> 3202) AND (iTerminalType <> 3204))	THEN
		bError		:= TRUE;
		iErrorId	:= 16#8002;
		iStep		:= 160;
	END_IF

(*-----------------------------------------------------------------*)

100:(*jetzige Sensoreinstellung lesen: Register 32*)
	stOutData.iCtrl	:= 16#A0;	(*Register 32 Lesen*)

	IF stInData.iState = 16#A0 THEN
		wReg32			:= INT_TO_WORD(stInData.iDataIn);
		A_SetConfigTable;		(*entsprechende Bits für den zu schreibenden Wert setzen, der Rest bleibt unberührt*)
		iStep:=110;
		IF	bSetConfigError	THEN
			iStep:=150;
		END_IF
	END_IF

110:(*Codewort Register 31 setzen: 16#1235 -> Schreibschutz aufheben*)
	stOutData.iCtrl	:= 16#DF;	(*Register 31 beschreiben*)
	stOutData.iDataOut	:= 16#1235;	(*Nutzdaten: Codewort*)

	IF stInData.iState = 16#9F THEN
		stOutData.iCtrl	:= 16#9F;	(*Register 31 Auslesen*)
		iStep:=120;
	END_IF

120:(*Bestätigung Codewort gesetzt erfragen*)
	IF	stInData.iDataIn	= 16#1235	THEN
		iStep:=130;
	END_IF

130:(*Nun Register 32 mit dem neuen Wert beschreiben*)
	stOutData.iCtrl	:= 16#E0;	(*Register 32 beschreiben*)
	stOutData.iDataOut	:= WORD_TO_INT(wSetReg32);

	IF stInData.iState = 16#A0 THEN
		iStep:=140;
	END_IF

140:(*Codewort Register 31 löschen: 16#0000 -> Schreibschutz setzen*)
	stOutData.iCtrl	:= 16#DF;	(*Register 31 beschreiben*)
	stOutData.iDataOut	:= 16#0000;

	IF stInData.iState = 16#9F THEN
		iStep:=150;
	END_IF

150:(*nach erfolgter Parametrierung Sensoreinstellung lesen: Register 32*)
	stOutData.iCtrl	:= 16#A0;	(*Register 32 Lesen*)

	IF stInData.iState = 16#A0 THEN
		wReg32			:= INT_TO_WORD(stInData.iDataIn);
		A_ReadConfigTable;
		iStep:=160;
	END_IF

160:(*Registerkommunikation beenden*)
	stOutData.iCtrl	:= 0; (*auch alle anderen Steuerbits mit ablöschen*)
	(*Rückmeldeabfrage Prozessdatenaustausch (Bit7) noch aktiv? *)
	(*alle anderen Bits könnten durch einen bestimmten Signalpegel gesetzt sein *)
	IF stInData.iState.7 = FALSE THEN
		iStep:=0;
	END_IF

END_CASE
END_FUNCTION_BLOCK
ACTION A_ReadConfigTable:
CASE (SHR(wReg32,12)) OF	(*Check sensor-type via the 4 most significant bits*)
	2#0000: sSensorType:='PT100';
	2#0001: sSensorType:='NI100';
	2#0010: sSensorType:='PT1000';
	2#0011: sSensorType:='PT500';
	2#0100: sSensorType:='PT200';
	2#0101: sSensorType:='NI1000';
	2#0110: sSensorType:='NI120';
	
	2#1110: sSensorType:='10Ohm .. 5000Ohm';
	2#1111: sSensorType:='10Ohm .. 1200Ohm';
ELSE
	sSensorType	:='Unknown';
	bError		:= TRUE;
	iErrorId	:= 16#802A;
END_CASE

bTwoWiredConnection:=wReg32.10;
END_ACTION
ACTION A_SetConfigTable:
bSetConfigError	:= FALSE;

wSetReg32:=wReg32 AND 2#0000111111111111;(*First clear the first 4 bits*)

CASE iSetSensorType OF	(*Then set the sensor-type via the 4 most significant bits - Bit 10 sets 2-wired-connection*)

	0:	wSetReg32:=wSetReg32 OR 2#0000000000000000;(*PT100*)
		wSetReg32.10:=FALSE;					(*1-Wired*)

	1:	wSetReg32:=wSetReg32 OR 2#0001000000000000;(*NI100*)
		wSetReg32.10:=FALSE;					(*1-Wired*)

	2:	wSetReg32:=wSetReg32 OR 2#0010000000000000;(*PT1000*)
		wSetReg32.10:=FALSE;					(*1-Wired*)

	3:	wSetReg32:=wSetReg32 OR 2#0011000000000000;(*PT500*)
		wSetReg32.10:=FALSE;					(*1-Wired*)

	4:	wSetReg32:=wSetReg32 OR 2#0100000000000000;(*PT200*)
		wSetReg32.10:=FALSE;					(*1-Wired*)

	5:	wSetReg32:=wSetReg32 OR 2#0101000000000000;(*NI1000*)
		wSetReg32.10:=FALSE;					(*1-Wired*)

	6:	wSetReg32:=wSetReg32 OR 2#0110000000000000;(*NI120*)
		wSetReg32.10:=FALSE;					(*1-Wired*)

	7:	wSetReg32:=wSetReg32 OR 2#1110000000000000;(*10Ohm .. 5000Ohm*)
		wSetReg32.10:=FALSE;					(*1-Wired*)

	8:	wSetReg32:=wSetReg32 OR 2#1111000000000000;(*10Ohm .. 1200Ohm*)
		wSetReg32.10:=FALSE;					(*1-Wired*)

	9:	wSetReg32:=wSetReg32 OR 2#0010000000000000;(*PT1000*)
		wSetReg32.10:=TRUE;						(*2-Wired*)

		IF (iTerminalType=3204)	THEN			(*2-Wired is not allowed for KL3204*)
			bSetConfigError	:= TRUE;
			bError			:= TRUE;
			iErrorId		:= 16#8028;
		END_IF
ELSE
	bSetConfigError	:= TRUE;
	bError			:= TRUE;
	iErrorId		:= 16#8029;
END_CASE
END_ACTION

(* POU FB_KL3228Config, ST *)
FUNCTION_BLOCK FB_KL3228Config
VAR_INPUT
	bConfigurate		: BOOL; 		(*Rising edge starts configuration including read-configuration afterwards*)
	bReadConfig			: BOOL;			(*Rising edge reads the actual configuration*)
	iSetSensorType		: INT;			(*Sensor-type to be set, see table*)
	tTimeout			: TIME :=t#5s;	(*Time-out-time for Reading/Configuration - initially set to 5s*)
END_VAR
VAR_OUTPUT
	bBusy				: BOOL;			(*Reading or configuration is in progress*)
	bError				: BOOL;			(*Error while reading/configuration*)
	iErrorId			: UDINT;		(*Id of the last upcoming error*)
	iState				: USINT;		(*As long as the funcion-block is not busy, this variable shows the state of the terminal, otherwise it is 0*)
	iDataIn				: INT;			(*As long as the funcion-block is not busy, this variable shows the dataIn of the terminal, otherwise it keeps the value previous to reding/configuration*)
	iTerminalType		: WORD;			(*Terminal-type-number, in this case 3228*)
	iSpecialType		: WORD;			(*Sub-type-number*)
	iFirmwareVersion	: WORD;			(*Firmware in ASCII-code*)
	sDescription		: STRING;		(*Terminal-type, special-type and firmware-version as readable text*)
	sSensorType			: STRING;		(*Text-description of entered sensor-type*)
END_VAR
VAR
	rtRead				: R_TRIG;
	rtSet				: R_TRIG;
	bSetReq				: BOOL;
	tonTimeout			: TON;
	iStep				: INT;
	bSetConfigError		: BOOL;
	wReg32				: WORD;
	wSetReg32			: WORD;
	wFirmware			: WORD;
	pFirmware			: POINTER TO WORD;
	sFirmware			: STRING(2);
	iDataInSaved		: INT;
END_VAR
VAR_IN_OUT
	stInData   			: ST_KL3228InData;	(* Process image of the inputs. *)
	stOutData 			: ST_KL3228OutData;	(* Process image of the outputs. *)
END_VAR
tonTimeout	(PT:=tTimeout);
IF	tonTimeout.Q	THEN
	bError			:= TRUE;
	iErrorId		:= 16#8001;
	iStep			:= 0;
END_IF

rtSet	(CLK:=bConfigurate);
rtRead	(CLK:=bReadConfig);

IF	(rtSet.Q OR rtRead.Q)	AND NOT bBusy THEN
	bBusy			:= TRUE;
	bError			:= FALSE;
	iErrorId		:= 0;
	iDataInSaved	:= stInData.iDataIn;
	tonTimeout.IN	:= TRUE;
	iStep			:= 10;
	IF	rtSet.Q	THEN
		bSetReq	:= TRUE;
	END_IF
END_IF

IF bBusy THEN
	iDataIn		:= iDataInSaved;
	iState		:= 0;
ELSE
	iDataIn		:= stInData.iDataIn;
	iState		:= stInData.iState;
END_IF


CASE iStep OF

0:	(*idle*)
	bBusy				:= FALSE;
	bSetReq				:= FALSE;
	tonTimeout.IN		:= FALSE;

10:	(*Klemmentyp (Kl32xx) auslesen: Register 8*)
	stOutData.iCtrl	:= 16#88;	(*Register 8 Lesen*)

	IF stInData.iState = 16#88 THEN
		iTerminalType	:= INT_TO_WORD(stInData.iDataIn);
		iStep:=20;
	END_IF

20:	(*Spezialtyp (Kl32xx-yyy) auslesen: Register 29*)
	stOutData.iCtrl	:= 16#9D;	(*Register 29 Lesen*)

	IF stInData.iState = 16#9D THEN
		iSpecialType	:= INT_TO_WORD(stInData.iDataIn);
		iStep:=30;
	END_IF

30:	(*Firmware auslesen: Register 9*)
	stOutData.iCtrl	:= 16#89;	(*Register 9 Lesen*)

	IF stInData.iState = 16#89 THEN
		iFirmwareVersion:= INT_TO_WORD(stInData.iDataIn);
		(*Umwandlung in STRING*)
		wFirmware		:= iFirmwareVersion;
		wFirmware		:= ROR(wFirmware,8);(*Reihenfolge der beiden Zeichen der Firmware tauschen*)
		pFirmware		:= ADR(sFirmware);	(*Einen Pointer auf den Info-String (Ausgang) legen*)
		pFirmware^		:= wFirmware;		(*Diesen Adressbereich mit dem richtig getauschen Wert beschreiben - damit ist auch der String beschrieben*)

		sDescription	:= CONCAT('Terminal ',WORD_TO_STRING(iTerminalType));

		CASE LEN(WORD_TO_STRING(iSpecialType)) OF
			1: sDescription	:= CONCAT(sDescription,'-000');
			2: sDescription	:= CONCAT(sDescription,'-00');
			3: sDescription	:= CONCAT(sDescription,'-0');
		ELSE
			sDescription	:= CONCAT(sDescription,'-');
		END_CASE

		sDescription	:= CONCAT(sDescription,WORD_TO_STRING(iSpecialType));
		sDescription	:= CONCAT(sDescription,' / Firmware ');
		sDescription	:= CONCAT(sDescription,sFirmware);

		IF bSetReq	THEN
			iStep:=100;
		ELSE
			iStep:=150;
		END_IF
	END_IF

	(*Falscher Klemmentyp angeschlossen, Konfiguration vorzeitig abbrechen*)
	IF (iTerminalType <> 3228)	THEN
		bError		:= TRUE;
		iErrorId	:= 16#8002;
		iStep		:= 160;
	END_IF

(*-----------------------------------------------------------------*)

100:(*jetzige Sensoreinstellung lesen: Register 32*)
	stOutData.iCtrl	:= 16#A0;	(*Register 32 Lesen*)

	IF stInData.iState = 16#A0 THEN
		wReg32			:= INT_TO_WORD(stInData.iDataIn);
		A_SetConfigTable;		(*entsprechende Bits für den zu schreibenden Wert setzen, der Rest bleibt unberührt*)
		iStep:=110;
		IF	bSetConfigError	THEN
			iStep:=150;
		END_IF
	END_IF

110:(*Codewort Register 31 setzen: 16#1235 -> Schreibschutz aufheben*)
	stOutData.iCtrl	:= 16#DF;	(*Register 31 beschreiben*)
	stOutData.iDataOut	:= 16#1235;	(*Nutzdaten: Codewort*)

	IF stInData.iState = 16#9F THEN
		stOutData.iCtrl	:= 16#9F;	(*Register 31 Auslesen*)
		iStep:=120;
	END_IF

120:(*Bestätigung Codewort gesetzt erfragen*)
	IF	stInData.iDataIn	= 16#1235	THEN
		iStep:=130;
	END_IF

130:(*Nun Register 32 mit dem neuen Wert beschreiben*)
	stOutData.iCtrl	:= 16#E0;	(*Register 32 beschreiben*)
	stOutData.iDataOut	:= WORD_TO_INT(wSetReg32);

	IF stInData.iState = 16#A0 THEN
		iStep:=140;
	END_IF

140:(*Codewort Register 31 löschen: 16#0000 -> Schreibschutz setzen*)
	stOutData.iCtrl	:= 16#DF;	(*Register 31 beschreiben*)
	stOutData.iDataOut	:= 16#0000;

	IF stInData.iState = 16#9F THEN
		iStep:=150;
	END_IF

150:(*nach erfolgter Parametrierung Sensoreinstellung lesen: Register 32*)
	stOutData.iCtrl	:= 16#A0;	(*Register 32 Lesen*)

	IF stInData.iState = 16#A0 THEN
		wReg32			:= INT_TO_WORD(stInData.iDataIn);
		A_ReadConfigTable;
		iStep:=160;
	END_IF

160:(*Registerkommunikation beenden*)
	stOutData.iCtrl	:= 0; (*auch alle anderen Steuerbits mit ablöschen*)
	(*Rückmeldeabfrage Prozessdatenaustausch (Bit7) noch aktiv? *)
	(*alle anderen Bits könnten durch einen bestimmten Signalpegel gesetzt sein *)
	IF stInData.iState.7 = FALSE THEN
		iStep:=0;
	END_IF

END_CASE
END_FUNCTION_BLOCK
ACTION A_ReadConfigTable:
CASE (SHR(wReg32,12)) OF	(*Check sensor-type via the 4 most significant bits*)
	2#0000: sSensorType	:= 'PT1000';
	2#0001: sSensorType	:= 'NI1000';
	2#0010: sSensorType	:= 'RSNI1000';
ELSE
	sSensorType	:='Unknown';
	bError		:= TRUE;
	iErrorId	:= 16#8031;
END_CASE
END_ACTION
ACTION A_SetConfigTable:
bSetConfigError	:= FALSE;

CASE iSetSensorType OF	(*Then set the sensor-type via the 4 most significant bits*)
	0:	wSetReg32	:= wReg32		AND 2#0000111111111111;(*First clear the first 4 bits*)
		wSetReg32	:= wSetReg32	OR 2#0000000000000000;(*PT1000*)	(*Then set the sensor-type via the 4 most significant bits*)

	1:	wSetReg32	:= wReg32		AND 2#0000111111111111;(*First clear the first 4 bits*)
		wSetReg32	:= wSetReg32	OR 2#0001000000000000;(*NI1000*)	(*Then set the sensor-type via the 4 most significant bits*)

	2:	wSetReg32	:= wReg32		AND 2#0000111111111111;(*First clear the first 4 bits*)
		wSetReg32	:= wSetReg32	OR 2#0010000000000000;(*RSNI1000*)(*Then set the sensor-type via the 4 most significant bits*)
ELSE
	bSetConfigError	:= TRUE;
	bError			:= TRUE;
	iErrorId		:= 16#8030;
END_CASE
END_ACTION
